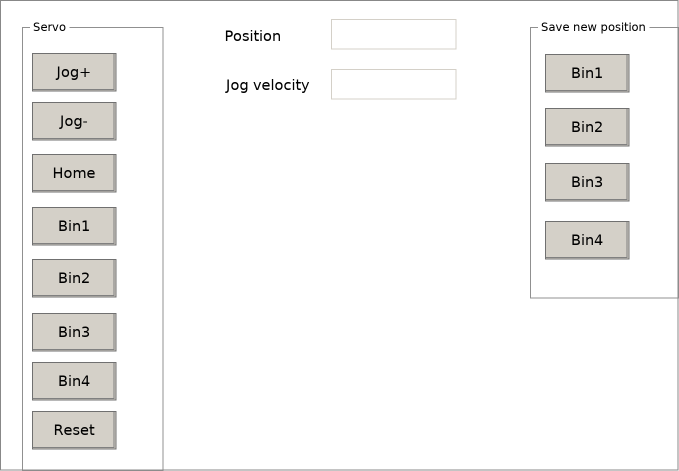
VISUALIZATION ServoMotionScreen  // 679x471
    GroupBox (22,19 141x452), "Servo"
        Button (10,34 84x38), "Jog+"
        Button (10,83 84x38), "Jog-"
        Button (10,135 84x38), "Home"
        Button (10,188 84x38), "Bin1"
        Button (10,240 84x38), "Bin2"
        Button (10,294 84x38), "Bin3"
        Button (10,343 84x38), "Bin4"
        Button (10,392 84x38), "Reset"
    Label (212,21 82x30), "Position"
    Label (212,70 112x30), "Jog velocity"
    Textfield (331,19 125x30)
    Textfield (331,69 125x30)
    GroupBox (530,19 149x279), "Save new position"
        Button (15,35 84x38), "Bin1"
        Button (15,89 84x38), "Bin2"
        Button (15,144 84x38), "Bin3"
        Button (15,202 84x38), "Bin4"
END_VISUALIZATION

(* stored: Version 1.1.0.1, ProductVersion 3.1.4024.13
   Visu ServoMotionScreen: Id {061a066e-eb74-49b5-a389-cec1d8a7b7a4} *)
